Staubli VAL3: start.pgx

program start()
  local string l_sKey
begin
  while size(sOrig)>8
    l_sKey=first(sOrig)
    delete(sOrig[l_sKey])
  endWhile

//  if first(sOrig)==""
//    delete(sTarget["Key1"])
//    popUpMsg("空")
//  else
//    popUpMsg(toString("",size(sOrig)))
//  endIf


   // popUpMsg(toString("",size(sTarget)))


end
